// TIA Portal project "Cau1" (V16)

(* hardware
DEVICE "S7-1200 station_1"  S7-1200 Station
   slot 0: "Rack_0"  S7-1200 Rack  Rack  V1.0
   slot 1: "PLC_1"  CPU 1212C DC/DC/DC  6ES7 212-1AE40-0XB0  V4.3
   slot 2: "DI 16/DQ 16x24VDC_1"  6ES7 223-1BL32-0XB0  V2.0
   slot 3: "DQ 16xRelay_1"  SM 1222 DQ16 x relay  6ES7 222-1HH32-0XB0  V2.0
*)

// ===== PLC "PLC_1"  CPU 1212C DC/DC/DC =====

VAR_GLOBAL   // PLC tag table "Default tag table"
   "A (NO)" AT %I0.5 : Bool;
   "KM1" AT %Q0.0 : Bool;
   "A (NC)" AT %I0.0 : Bool;
   "Biến giữ KM1" AT %M0.1 : Bool;
   "Biến giữ KM2" AT %M0.2 : Bool;
   "Biến giữ KM3" AT %M0.3 : Bool;
   "B (NC)" AT %I0.1 : Bool;
   "C (NC)" AT %I0.2 : Bool;
   "Biến giữ KM4" AT %M0.4 : Bool;
   "D (NC)" AT %I0.3 : Bool;
   "Biến giữ KM5" AT %M0.5 : Bool;
   "E (NC)" AT %I0.4 : Bool;
   "Start" AT %I1.3 : Bool;
   "Stop" AT %I1.2 : Bool;
   "B (NO)" AT %I0.6 : Bool;
   "C (NO)" AT %I0.7 : Bool;
   "D (NO)" AT %I8.0 : Bool;
   "E (NO)" AT %I8.1 : Bool;
   "KM2" AT %Q0.1 : Bool;
   "KM3" AT %Q0.2 : Bool;
   "KM4" AT %Q0.3 : Bool;
   "KM5" AT %Q0.4 : Bool;
END_VAR

ORGANIZATION_BLOCK "Main"   // OB1, LAD, ProgramCycle
TITLE = "Main Program Sweep (Cycle)"
{ S7_Optimized_Access := 'TRUE' }
VERSION : 0.1
   VAR_INPUT
      Initial_Call : Bool;   // Initial call of this OB
      Remanence : Bool;   // =True, if remanent data are available
   END_VAR
BEGIN

REGION Network 1
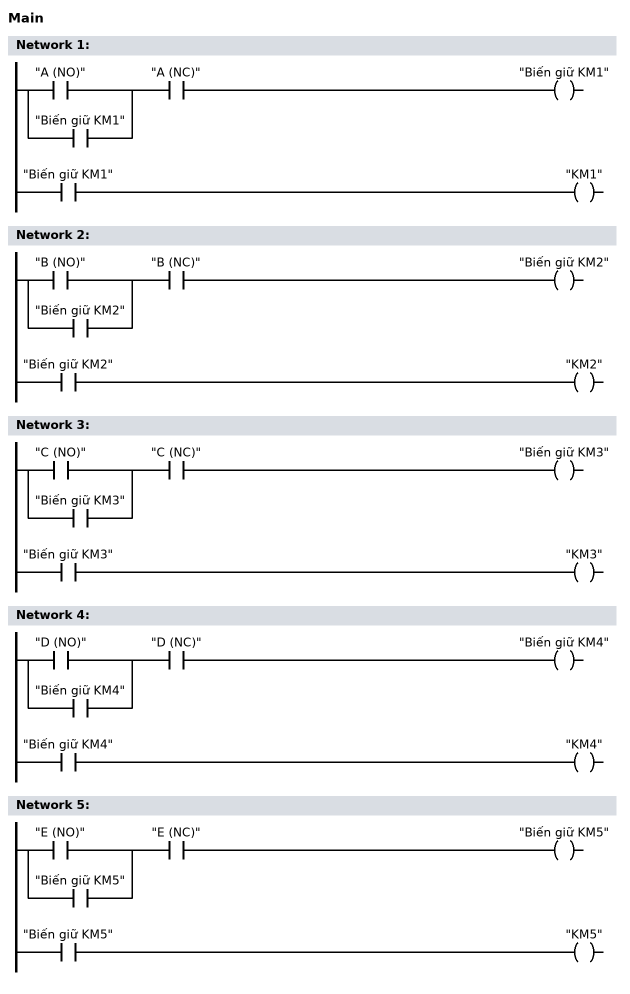
   RUNG wire#powerrail
      Contact( "A (NO)" )
      wire#w1
      Contact( "A (NC)" )
      Coil( "Biến giữ KM1" )
   END_RUNG
   RUNG wire#powerrail
      Contact( "Biến giữ KM1" )
   END_RUNG wire#w1
   RUNG wire#powerrail
      Contact( "Biến giữ KM1" )
      Coil( "KM1" )
   END_RUNG
   // the same network as SCL:
   "Biến giữ KM1" := ("A (NO)" OR "Biến giữ KM1") AND "A (NC)";
   "KM1" := "Biến giữ KM1";
END_REGION

REGION Network 2
   RUNG wire#powerrail
      Contact( "B (NO)" )
      wire#w1
      Contact( "B (NC)" )
      Coil( "Biến giữ KM2" )
   END_RUNG
   RUNG wire#powerrail
      Contact( "Biến giữ KM2" )
   END_RUNG wire#w1
   RUNG wire#powerrail
      Contact( "Biến giữ KM2" )
      Coil( "KM2" )
   END_RUNG
   // the same network as SCL:
   "Biến giữ KM2" := ("B (NO)" OR "Biến giữ KM2") AND "B (NC)";
   "KM2" := "Biến giữ KM2";
END_REGION

REGION Network 3
   RUNG wire#powerrail
      Contact( "C (NO)" )
      wire#w1
      Contact( "C (NC)" )
      Coil( "Biến giữ KM3" )
   END_RUNG
   RUNG wire#powerrail
      Contact( "Biến giữ KM3" )
   END_RUNG wire#w1
   RUNG wire#powerrail
      Contact( "Biến giữ KM3" )
      Coil( "KM3" )
   END_RUNG
   // the same network as SCL:
   "Biến giữ KM3" := ("C (NO)" OR "Biến giữ KM3") AND "C (NC)";
   "KM3" := "Biến giữ KM3";
END_REGION

REGION Network 4
   RUNG wire#powerrail
      Contact( "D (NO)" )
      wire#w1
      Contact( "D (NC)" )
      Coil( "Biến giữ KM4" )
   END_RUNG
   RUNG wire#powerrail
      Contact( "Biến giữ KM4" )
   END_RUNG wire#w1
   RUNG wire#powerrail
      Contact( "Biến giữ KM4" )
      Coil( "KM4" )
   END_RUNG
   // the same network as SCL:
   "Biến giữ KM4" := ("D (NO)" OR "Biến giữ KM4") AND "D (NC)";
   "KM4" := "Biến giữ KM4";
END_REGION

REGION Network 5
   RUNG wire#powerrail
      Contact( "E (NO)" )
      wire#w1
      Contact( "E (NC)" )
      Coil( "Biến giữ KM5" )
   END_RUNG
   RUNG wire#powerrail
      Contact( "Biến giữ KM5" )
   END_RUNG wire#w1
   RUNG wire#powerrail
      Contact( "Biến giữ KM5" )
      Coil( "KM5" )
   END_RUNG
   // the same network as SCL:
   "Biến giữ KM5" := ("E (NO)" OR "Biến giữ KM5") AND "E (NC)";
   "KM5" := "Biến giữ KM5";
END_REGION
END_ORGANIZATION_BLOCK